// TIA Portal V16 export
// export: Created 2021-03-04T22:04:03.1808656Z, ExportSetting WithDefaults, DisplayName Totally Integrated Automation Portal, DisplayVersion V16, DisplayName TIA Portal Version Control Interface, DisplayVersion V16, DisplayName TIA Portal Openness, DisplayVersion V16, DisplayName SINAMICS Startdrive Advanced, DisplayVersion V16, DisplayName SINAMICS Startdrive G130, G150, S120, S150, SINAMICS MV, S210, DisplayVersion V16, DisplayName SINAMICS Startdrive G110M, G120, G120C, G120D, G120P, DisplayVersion V16, DisplayName STEP 7 Professional, DisplayVersion V16, DisplayName STEP 7 Safety, DisplayVersion V16, DisplayName WinCC Professional, DisplayVersion V16
FUNCTION "fcHMIBitEnable" : Void   // FC329, LAD
TITLE = Handles an async reading of an HMI bit to avoid race conditions, includes an enable bit
{ S7_Optimized_Access := 'TRUE' }
VERSION : 0.1
// stored: AutoNumber true, IsIECCheckEnabled false, SetENOAutomatically false, UDAEnableTagReadback false
   VAR_INPUT
      bInToggle : Bool;
      bInLatch : Bool;
      bInEnable : Bool;
   END_VAR
   VAR_OUTPUT
      bOutEnable : Bool;
   END_VAR
   VAR_IN_OUT
      bInOutHMI : Bool;
      bInOutPLC : Bool;
   END_VAR
   VAR_TEMP   // added for the SCL form of the ladder/FBD networks
      _w1 : Bool;
   END_VAR
BEGIN

REGION Network 1: If not latching or toggling, reset the PLC bit every scan
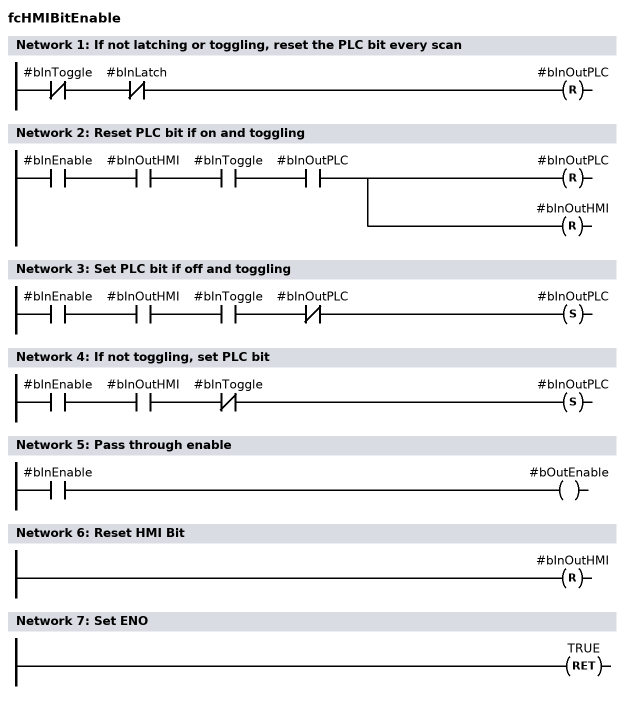
   RUNG wire#powerrail
      I_Contact( #bInToggle )
      I_Contact( #bInLatch )
      R_Coil( #bInOutPLC )
   END_RUNG
   // the same network as SCL:
   IF NOT #bInToggle AND NOT #bInLatch THEN #bInOutPLC := FALSE; END_IF;
END_REGION

REGION Network 2: Reset PLC bit if on and toggling
   RUNG wire#powerrail
      Contact( #bInEnable )
      Contact( #bInOutHMI )
      Contact( #bInToggle )
      Contact( #bInOutPLC )
      wire#w1
      R_Coil( #bInOutPLC )
   END_RUNG
   RUNG wire#w1
      R_Coil( #bInOutHMI )
   END_RUNG
   // the same network as SCL:
   #_w1 := #bInEnable AND #bInOutHMI AND #bInToggle AND #bInOutPLC;
   IF #_w1 THEN
       #bInOutPLC := FALSE;
       #bInOutHMI := FALSE;
   END_IF;
END_REGION

REGION Network 3: Set PLC bit if off and toggling
   RUNG wire#powerrail
      Contact( #bInEnable )
      Contact( #bInOutHMI )
      Contact( #bInToggle )
      I_Contact( #bInOutPLC )
      S_Coil( #bInOutPLC )
   END_RUNG
   // the same network as SCL:
   IF #bInEnable AND #bInOutHMI AND #bInToggle AND NOT #bInOutPLC THEN #bInOutPLC := TRUE; END_IF;
END_REGION

REGION Network 4: If not toggling, set PLC bit
   RUNG wire#powerrail
      Contact( #bInEnable )
      Contact( #bInOutHMI )
      I_Contact( #bInToggle )
      S_Coil( #bInOutPLC )
   END_RUNG
   // the same network as SCL:
   IF #bInEnable AND #bInOutHMI AND NOT #bInToggle THEN #bInOutPLC := TRUE; END_IF;
END_REGION

REGION Network 5: Pass through enable
   RUNG wire#powerrail
      Contact( #bInEnable )
      Coil( #bOutEnable )
   END_RUNG
   // the same network as SCL:
   #bOutEnable := #bInEnable;
END_REGION

REGION Network 6: Reset HMI Bit
   RUNG wire#powerrail
      R_Coil( #bInOutHMI )
   END_RUNG
   // the same network as SCL:
   #bInOutHMI := FALSE;
END_REGION

REGION Network 7: Set ENO
   RUNG wire#powerrail
      ReturnCoil( TRUE )
   END_RUNG
   // the same network as SCL:
   ENO := TRUE;
   RETURN;
END_REGION
END_FUNCTION
